ABB RobotStudio station: medicine_dispatcher_part2.rspag

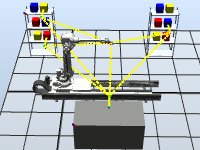
--- station ---
Station Examen (saved by RobotStudio 6.8.8307.1040)
Controller Sistema1, task T_ROB1: task frame (RAPID world) sits at (0, 0, 397.5) mm in the station
Controller Sistema1
  mechanical unit ROB_1: IRB4600_20_250_C_01, 6 joints, base frame (0, 0, 0) mm
  mechanical unit TRACK: RTT_Bobin_2_7, 1 joints, base frame (0, 0, 0) mm
Layout (positions relative to the parent item):
  - IRB4600_20_250_C_01 [mechanism, from Robots\IRB4600_20_250_C_G_01.rslib] at (0, 0, 397.5) mm; joint values [0, 0, 0, 0, 0.5236, 0] (rad or m)
  - RTT_Bobin_2_7 [mechanism] at (0, 0, 0) mm; joint values [0] (rad or m)
      links: Base, Link1
  - Estante1 [graphiccomponentgroup, from Libraries\Estante.rslib] at (-500, 2000, 0) mm
    - stojna [part, from Libraries\Estante.rslib]
    - police [part, from Libraries\Estante.rslib] at (-500, 200, 124) mm
    - stojna [part, from Libraries\Estante.rslib] at (0, 400, 0) mm, rotated rx 0 ry 0 rz 90 deg
    - stojna [part, from Libraries\Estante.rslib] at (-1000, 400, 0) mm, rotated rx 0 ry 0 rz 180 deg
    - stojna [part, from Libraries\Estante.rslib] at (-1000, 0, 0) mm, rotated rx 0 ry 0 rz -90 deg
    - police [part, from Libraries\Estante.rslib] at (-500, 200, 721) mm
    - police [part, from Libraries\Estante.rslib] at (-500, 200, 1318) mm
    - police [part, from Libraries\Estante.rslib] at (-500, 200, 1915) mm
    - Caja Roja2 [part, from Libraries\Estante.rslib] at (-800, 125, 1321.04) mm
    - Caja Azul2 [part, from Libraries\Estante.rslib] at (-800, 125, 1918.04) mm
    - Caja Amarilla2 [part, from Libraries\Estante.rslib] at (-800, 125, 724.04) mm
    - Caja Roja1 [part, from Libraries\Estante.rslib] at (-450, 125, 724.04) mm
    - Caja Amarilla1 [part, from Libraries\Estante.rslib] at (-450, 125, 1918.04) mm
    - Caja Azul1 [part, from Libraries\Estante.rslib] at (-450, 125, 1321.04) mm
  - Estante2 [graphiccomponentgroup, from Libraries\Estante.rslib] at (4000, 2000, 0) mm
    - stojna [part, from Libraries\Estante.rslib]
    - police [part, from Libraries\Estante.rslib] at (-500, 200, 124) mm
    - stojna [part, from Libraries\Estante.rslib] at (0, 400, 0) mm, rotated rx 0 ry 0 rz 90 deg
    - stojna [part, from Libraries\Estante.rslib] at (-1000, 400, 0) mm, rotated rx 0 ry 0 rz 180 deg
    - stojna [part, from Libraries\Estante.rslib] at (-1000, 0, 0) mm, rotated rx 0 ry 0 rz -90 deg
    - police [part, from Libraries\Estante.rslib] at (-500, 200, 721) mm
    - police [part, from Libraries\Estante.rslib] at (-500, 200, 1318) mm
    - police [part, from Libraries\Estante.rslib] at (-500, 200, 1915) mm
    - Caja Roja2 [part, from Libraries\Estante.rslib] at (-800, 125, 1321.04) mm
    - Caja Azul2 [part, from Libraries\Estante.rslib] at (-800, 125, 1918.04) mm
    - Caja Amarilla2 [part, from Libraries\Estante.rslib] at (-800, 125, 724.04) mm
    - Caja Roja1 [part, from Libraries\Estante.rslib] at (-450, 125, 724.04) mm
    - Caja Amarilla1 [part, from Libraries\Estante.rslib] at (-450, 125, 1918.04) mm
    - Caja Azul1 [part, from Libraries\Estante.rslib] at (-450, 125, 1321.04) mm
  - Succionador [smart component] at (1479.11, 0, 2120) mm, rotated rx 180 ry 60 rz 180 deg
      signals: DI SuctionON, DO Detach
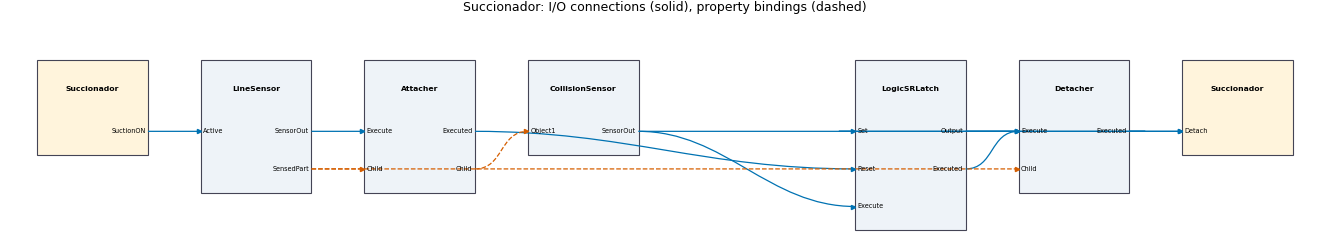
      connections:
        Succionador.SuctionON -> LineSensor.Active
        LogicSRLatch.Output -> Succionador.Detach
        LogicGate.Output -> Detacher.Execute
        LineSensor.SensorOut -> Attacher.Execute
        Detacher.Executed -> LogicSRLatch.Set
        Attacher.Executed -> LogicSRLatch.Reset
        Positioner.Executed -> Detacher.Execute
        CollisionSensor.SensorOut -> Positioner.Execute
        CollisionSensor.SensorOut -> Detacher.Execute
        Detacher.Executed -> Succionador.Detach
        LineSensor.SensedPart => Attacher.Child
        LineSensor.SensedPart => Detacher.Child
        Attacher.Child => CollisionSensor.Object1
    - Chupon [mechanism, from Libraries\Chupon4600.rslib] at (0, 0, 0) mm
    - LineSensor [smart component, from Components\LineSensor.rslib]
        properties: Start=[0 0 0.107]; End=[0 0 0.155]; Radius=0.002; SensedPart=(none); SensedPoint=[0 0 0]
      - _sensorPart_ [part]
    - Attacher [smart component, from Components\Attacher.rslib]
        properties: Parent=Chupon; Flange=0; Child=(none); Mount=false; Offset=[0 0 0]; Orientation=[0 0 0]
    - Detacher [smart component, from Components\Detacher.rslib]
        properties: Child=(none); KeepPosition=true
    - CollisionSensor [smart component, from Components\CollisionSensor.rslib]
        properties: Object1=(none); Object2=Pieza_2; NearMiss=0.001; Part1=(none); Part2=(none); CollisionType=0
  - Mesa [part, from Libraries\Mesa.rslib]
  - Pieza_2 [part]
Attachment: Chupon is attached to IRB4600_20_250_C_01 / Link6
Attachment: IRB4600_20_250_C_01 is attached to RTT_Bobin_2_7 / Link1
Attachment: Succionador is attached to IRB4600_20_250_C_01 / Link6
Station signals: DI Caja1, DI Caja2, DI Caja3
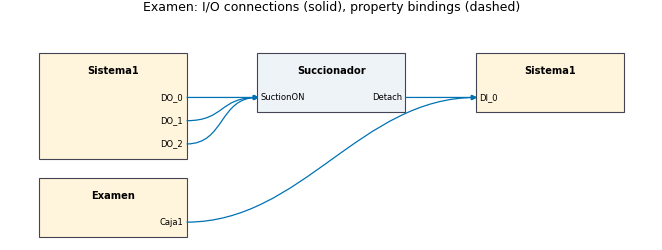
Station logic (signal -> signal, property => property):
  Sistema1.DO_0 -> Succionador.SuctionON
  Sistema1.DO_1 -> Succionador.SuctionON
  Sistema1.DO_2 -> Succionador.SuctionON
  Examen.Caja1 -> Sistema1.DI_0
  Succionador.Detach -> Sistema1.DI_0

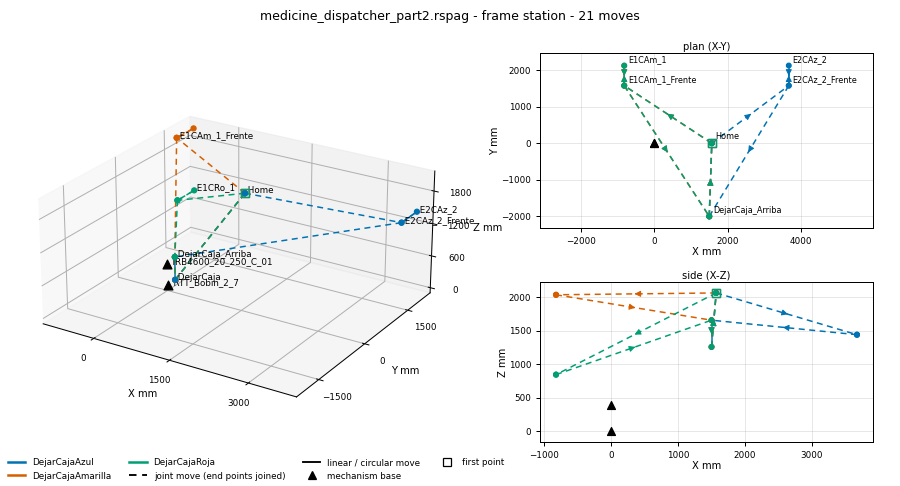
[picture p0: tool path of medicine_dispatcher_part2.rspag in frame station, 21 of 21 moves have a stored position in this frame; points joined in program order, loops and branches not executed]
--- Backups/Sistema1/RAPID/TASK1/PROGMOD/CalibData.mod ---
MODULE CalibData
	PERS tooldata Chupon:=[TRUE,[[0,0,105],[1,0,0,0]],[1,[0,0,1],[1,0,0,0],0,0,0]];
	TASK PERS wobjdata Estante1:=[FALSE,TRUE,"",[[-1496,2004,1517.5],[1,0,0,0]],[[0,0,0],[1,0,0,0]]];
	TASK PERS wobjdata Estante2:=[FALSE,TRUE,"",[[0,0,0],[1,0,0,0]],[[0,0,0],[1,0,0,0]]];
	TASK PERS wobjdata Mesa:=[FALSE,TRUE,"",[[500,-2500,602.5],[1,0,0,0]],[[0,0,0],[1,0,0,0]]];
ENDMODULE

--- Backups/Sistema1/RAPID/TASK1/PROGMOD/Module1.mod ---
MODULE Module1
	CONST robtarget Home:=[[1570.044826719,0,1670],[0.5,0,0.866025404,0],[0,0,0,0],[0,9E+09,9E+09,9E+09,9E+09,9E+09]];
	CONST robtarget E2CAz_2_Frente:=[[3675.00002564,1575.00005861,1045.499996445],[0.499999983,-0.500000004,0.500000007,0.500000006],[0,1,2,0],[2700,9E+09,9E+09,9E+09,9E+09,9E+09]];
	CONST robtarget E2CAz_2:=[[3675.00001464,2125.00005861,1045.499984345],[0.499999983,-0.500000004,0.500000007,0.500000006],[0,1,2,0],[2700,9E+09,9E+09,9E+09,9E+09,9E+09]];
	CONST robtarget DejarCaja_Arriba:=[[999.999806174,499.99999873,659.999985868],[0.00798397,-0.707061845,-0.707061568,-0.007983886],[-2,-1,-1,0],[1510.554985839,9E+09,9E+09,9E+09,9E+09,9E+09]];
	CONST robtarget DejarCaja:=[[999.999806174,499.99999873,259.999985868],[0.00798397,-0.707061845,-0.707061568,-0.007983886],[-2,-1,-1,0],[1510.554985839,9E+09,9E+09,9E+09,9E+09,9E+09]];
	CONST robtarget E1CAm_1_Frente:=[[670.999943993,-428.999956415,124.999999032],[0.499999973,-0.500000012,0.499999999,0.500000017],[1,-1,0,0],[0,9E+09,9E+09,9E+09,9E+09,9E+09]];
	CONST robtarget E1CAm_1:=[[671.00002689,117.000055454,124.999970405],[0.499999991,-0.499999916,0.499999992,0.500000101],[1,-2,1,0],[0,9E+09,9E+09,9E+09,9E+09,9E+09]];
	CONST robtarget E1CRo_1_Frente:=[[670.999969854,-428.999900879,-1068.999806594],[0.499999788,-0.49999955,0.500000338,0.500000324],[1,2,1,0],[0,9E+09,9E+09,9E+09,9E+09,9E+09]];
	CONST robtarget E1CRo_1:=[[671.000011571,118.999905382,-1068.999997128],[0.5,-0.50000001,0.499999978,0.500000012],[1,2,1,0],[0,9E+09,9E+09,9E+09,9E+09,9E+09]];
	PROC DejarCajaAzul()
	    MoveJ Home,v1000,z100,Chupon\WObj:=wobj0;
	    MoveJ E2CAz_2_Frente,v1000,z100,Chupon\WObj:=Estante2;
	    MoveJ E2CAz_2,v1000,z100,Chupon\WObj:=Estante2;
	    MoveL E2CAz_2_Frente,v1000,z100,Chupon\WObj:=Estante2;
	    MoveJ DejarCaja_Arriba,v1000,z100,Chupon\WObj:=Mesa;
	    MoveL DejarCaja,v1000,z100,Chupon\WObj:=Mesa;
		MoveJ Home,v1000,z100,Chupon\WObj:=wobj0;
	ENDPROC
	PROC DejarCajaAmarilla()
	    MoveJ Home,v1000,z100,Chupon\WObj:=wobj0;
	    MoveJ E1CAm_1_Frente,v1000,z100,Chupon\WObj:=Estante1;
	    MoveJ E1CAm_1,v1000,z100,Chupon\WObj:=Estante1;
	    MoveJ E1CAm_1_Frente,v1000,z100,Chupon\WObj:=Estante1;
	    MoveJ DejarCaja_Arriba,v1000,z100,Chupon\WObj:=Mesa;
	    MoveJ DejarCaja,v1000,z100,Chupon\WObj:=Mesa;
		MoveJ Home,v1000,z100,Chupon\WObj:=wobj0;
	ENDPROC
	PROC DejarCajaRoja()
	    MoveJ Home,v1000,z100,Chupon\WObj:=wobj0;
	    MoveJ E1CRo_1_Frente,v1000,z100,Chupon\WObj:=Estante1;
	    MoveJ E1CRo_1,v1000,z100,Chupon\WObj:=Estante1;
	    MoveJ E1CRo_1_Frente,v1000,z100,Chupon\WObj:=Estante1;
	    MoveJ DejarCaja_Arriba,v1000,z100,Chupon\WObj:=Mesa;
	    MoveJ DejarCaja,v1000,z100,Chupon\WObj:=Mesa;
	    MoveJ Home,v1000,z100,Chupon\WObj:=wobj0;
	ENDPROC
ENDMODULE

--- Backups/Sistema1/SYSPAR/EIO.cfg ---
EIO:CFG_1.0:6:1::
#
INDUSTRIAL_NETWORK:

      -Name "DeviceNet" -Label "DeviceNet Master/Slave Network" -Address "2"
#
DEVICENET_DEVICE:

      -Name "d652" -VendorName "ABB Robotics" -ProductName "24 VDC I/O Device"\
      -Label "DSQC 652 24 VDC I/O Device" -ProductCode 26 -DeviceType 7\
      -ConnectionType "COS" -OutputSize 2 -InputSize 2
#
DEVICENET_INTERNAL_DEVICE:

      -Name "DN_Internal_Device" -VendorName "ABB Robotics"\
      -ProductName "DeviceNet Internal Slave Device"
#
EIO_SIGNAL:

      -Name "DI_0" -SignalType "DI" -Device "d652" -DeviceMap "0" -Access "All"

      -Name "DI_1" -SignalType "DI" -Device "d652" -DeviceMap "1" -Access "All"

      -Name "DO_0" -SignalType "DO" -Device "d652" -DeviceMap "0" -Access "All"

      -Name "DO_1" -SignalType "DO" -Device "d652" -DeviceMap "1" -Access "All"

      -Name "DI_2" -SignalType "DI" -Device "d652" -DeviceMap "2" -Access "All"

      -Name "DO_2" -SignalType "DO" -Device "d652" -DeviceMap "2" -Access "All"
